Yaskawa INFORM job: S1_LOADING_POS_BATMAN.JBI

/JOB
//NAME S1_LOADING_POS_BATMAN
///FOLDERNAME OBROTNIK
//POS
///NPOS 0,0,0,0,0,0
//INST
///DATE 2023/11/17 09:33
///ATTR SC,RW,RJ
////FRAME ROBOT
///GROUP1 ST1
NOP
END
